RoboDK station: Maoyi_GlueDispensing_PM3.rdk

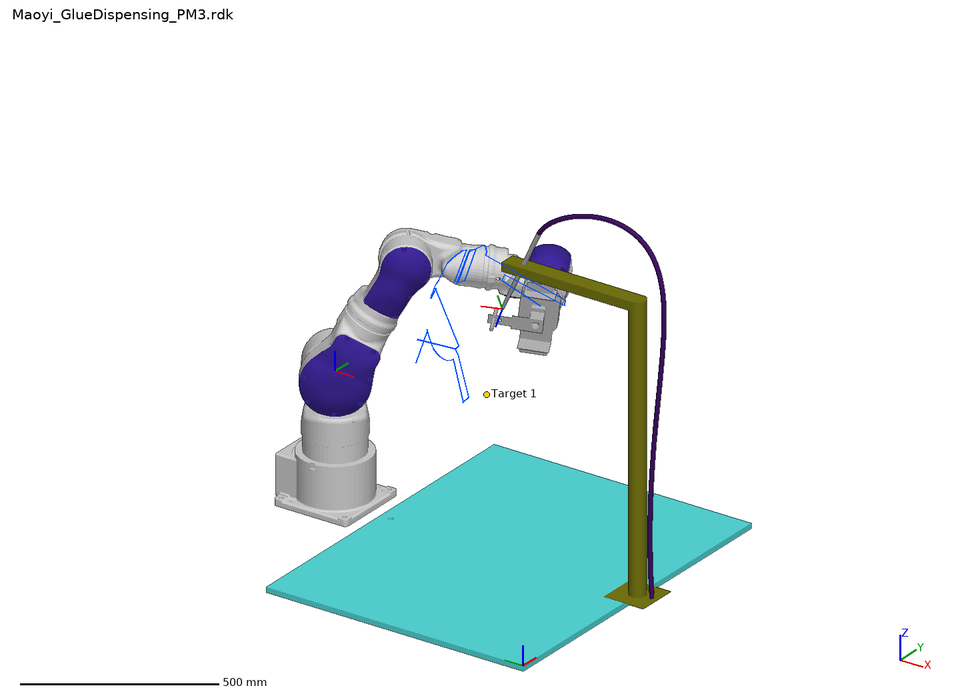
[picture v0: the station drawn from its stored meshes, robots at their saved joint values, targets as dots, program paths as lines]
Station Maoyi_GlueDispensing_PM3 (saved by RoboDK 5.2.1). Poses are relative to the parent item; angles as X-Y-Z fixed-axis rotations.
Station parameters (name, value as stored): IO_5, 1, IO_1, 0, IO_2, 0, IO_3, 1, CollisionFreePlanner, Motoman SIA10D, CollisionFreePlanner-Rob Motoman SIA10D
  - frame Motoman SIA10D Base at (0, 0, 360) mm
    - robot Motoman SIA10D: 7 axes, payload 10 kg, reach 720 mm, repeatability 0.1 mm, weight 60 kg
        modified DH rows (alpha deg, a mm, theta deg, d mm): 0, 0, 0, 360; -90, 0, 0, 0; 90, 0, 0, 360; -90, 0, 0, 0; 90, 0, 0, 360; -90, 0, 0, 0; 90, 0, 180, 155
        base shift (0, 0, -360) mm
        joint limits [-180, -110, -170, -135, -180, -110, -180] to [180, 110, 170, 135, 180, 110, 180]; home [0, 0, 0, 90, 0, 0, 0]; saved at [35.072, 29.67, 0, 66.212, -82.383, 96.989, -179.696]
      - tool Suction_cup, TCP at (106, 0, 141) mm, size 171 x 210 x 141 mm, geometry from Suction_cup.step
      - tool Path 1, TCP at (0, 0, 0) mm
    - frame Working plan at (927.5, -500, -365) mm, rotated rx 0 ry 0 rz 90 deg
      - object robot_platform1 at (0, 0, 0) mm, size 1000 x 790 x 15 mm, geometry from robot_platform1.step
      - object Dispensing Tool at (0, 0, 0) mm, rotated rx 90 ry 0 rz 180 deg, size 120 x 1028.7 x 505.5 mm, geometry from Dispensing Tool.step
      - target Target 1 (Cartesian target) at (500, 461.5, 429) mm, rotated rx -180 ry 0 rz -90 deg; joints [0, 0, 0, 90, 0, 90, 0] of Motoman SIA10D
  - frame Glue at (512.5, 0, 678) mm, rotated rx 169 ry -15 rz -130 deg
  - machining project Path 1 Settings: rotZ(0) | rotX(0)*rotY(0) | rotz(0) | onStart | onPathStart | onApproach | onPoint | onRetract | onFinish | SetRPM(%1) | SetTool(%1) | Extruder(%1) | default | default | OutOnMov(%1) | OutOffMov(%1) | onPathFinish | M_RunCode(%1) | WAN Miniport (IPv6)-QoS 
  - program Path (93 instructions, listed below)
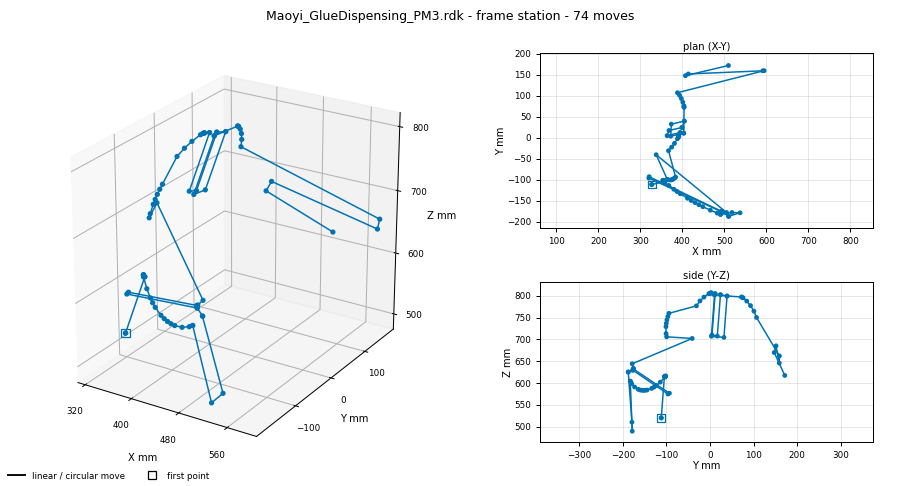
[picture p0: tool path of Maoyi_GlueDispensing_PM3.rdk in frame station, 74 of 74 moves have a stored position in this frame; points joined in program order, loops and branches not executed]

--- program Path (robot Motoman SIA10D) ---
  Smooth(1)
  Set speed (1000.0 mm/s)
  Set Ref.: Glue
  Set Tool: Path 1
  Show Path 1
  MoveJ 1 to (157.11, 29.72, 215.15) mm, rotated rx 0 ry 88 rz 170 deg; joints [-43.735, 4.404, 0, 111.833, 70.327, 95.789, -105.561]
  MoveL 2 to (157.11, 29.72, 215.15) mm, rotated rx 0 ry 88 rz 170 deg; joints [-43.735, 4.404, 0, 111.833, 70.327, 95.789, -105.561]
  MoveL 3 to (157.11, 29.72, 115.15) mm, rotated rx 0 ry 88 rz 170 deg; joints [-39.6, 2.361, 0, 98.055, 73.469, 96.968, -89.206]
  MoveL 4 to (157.11, 29.72, 115.15) mm, rotated rx 0 ry 88 rz 170 deg; joints [-39.6, 2.361, 0, 98.055, 73.469, 96.968, -89.206]
  Set speed (50.0 mm/s)
  MoveL 5 to (157.93, 34.33, 115.15) mm, rotated rx 0 ry 88 rz 170 deg; joints [-39.683, 1.614, 0, 98.657, 73.469, 97.088, -89.089]
  MoveL 6 to (157.93, 34.32, 115.15) mm, rotated rx 0 ry 88 rz 170 deg; joints [-39.683, 1.616, 0, 98.655, 73.469, 97.09, -89.09]
  MoveL 7 to (158.06, 34.91, 115.26) mm, rotated rx -2.73 ry 88 rz 167.24 deg; joints [-39.701, 1.529, 0, 98.739, 73.466, 97.13, -89.188]
  MoveL 8 to (158.06, 34.43, 115.85) mm, rotated rx -18.04 ry 87.9 rz 151.87 deg; joints [-39.727, 1.632, 0, 98.745, 73.448, 97.185, -89.858]
  MoveL 9 to (157.82, 32.09, 117.26) mm, rotated rx -45.21 ry 87.16 rz 124.55 deg; joints [-39.76, 2.054, 0, 98.615, 73.405, 97.245, -91.521]
  MoveL 10 to (154.79, 14.07, 124.94) mm, rotated rx -79.41 ry 79.05 rz 90.27 deg; joints [-39.761, 4.944, 0, 97.388, 73.212, 96.698, -101.87]
  MoveL 11 to (152.01, -2.22, 129.27) mm, rotated rx -83.67 ry 71.55 rz 85.94 deg; joints [-39.66, 7.569, 0, 95.743, 73.132, 96.266, -110.361]
  MoveL 12 to (150.39, -11.66, 130.72) mm, rotated rx -84.8 ry 67.34 rz 84.72 deg; joints [-39.564, 9.1, 0, 94.562, 73.121, 96.077, -114.908]
  MoveL 13 to (148.65, -21.63, 131.47) mm, rotated rx -85.59 ry 63.01 rz 83.78 deg; joints [-39.434, 10.743, 0, 93.127, 73.132, 95.975, -119.417]
  MoveL 14 to (145.06, -41.61, 130.64) mm, rotated rx -86.59 ry 54.07 rz 82.68 deg; joints [-39.109, 13.918, 0, 89.873, 73.23, 95.62, -128.205]
  MoveL 15 to (143.2, -51.74, 128.99) mm, rotated rx -86.92 ry 49.53 rz 82.27 deg; joints [-38.91, 15.538, 0, 87.958, 73.31, 95.519, -132.41]
  MoveL 16 to (141.35, -61.66, 126.55) mm, rotated rx -87.17 ry 45.01 rz 81.92 deg; joints [-38.694, 17.127, 0, 85.908, 73.408, 95.449, -136.437]
  MoveL 17 to (139.52, -71.34, 123.32) mm, rotated rx -87.37 ry 40.49 rz 81.63 deg; joints [-38.462, 18.685, 0, 83.728, 73.521, 95.41, -140.298]
  MoveL 18 to (137.59, -80.96, 119.31) mm, rotated rx -87.53 ry 35.95 rz 81.29 deg; joints [-38.204, 20.28, 0, 81.348, 73.653, 95.468, -144.012]
  MoveL 19 to (134.09, -98.51, 109.2) mm, rotated rx -87.76 ry 26.98 rz 80.87 deg; joints [-37.688, 23.195, 0, 76.452, 73.945, 95.527, -150.939]
  MoveL 20 to (131.11, -113.4, 97.08) mm, rotated rx -87.89 ry 18.43 rz 80.59 deg; joints [-37.184, 25.777, 0, 71.498, 74.251, 95.627, -157.067]
  MoveL 21 to (129.91, -120.19, 89.79) mm, rotated rx -87.94 ry 13.91 rz 80.57 deg; joints [-36.937, 26.977, 0, 68.888, 74.405, 95.615, -160.156]
  Set speed (1000.0 mm/s)
  MoveL 22 to (129.91, -120.19, 89.79) mm, rotated rx -87.94 ry 13.91 rz 80.57 deg; joints [-36.937, 26.977, 0, 68.888, 74.405, 95.615, -160.156]
  MoveL 23 to (79.99, -157.87, 189.79) mm, rotated rx -87.94 ry 13.91 rz 60.22 deg; joints [-33.756, 43.629, 0, 63.422, 72.969, 109.883, -171.1]
  Set speed (1000.0 mm/s)
  MoveL 24 to (73.82, -168.5, 164.19) mm, rotated rx -88 ry 0 rz 60.21 deg; joints [-32.838, 45.387, 0, 56.918, 74.962, 109.853, -179.878]
  MoveL 25 to (127, -133.09, 64.19) mm, rotated rx -88 ry 0 rz 80.21 deg; joints [-36.118, 29.852, 0, 61.258, 74.923, 95.954, -169.241]
  MoveL 26 to (126.52, -133.55, 64.19) mm, rotated rx -88 ry 0 rz 80 deg; joints [-36.071, 30.04, 0, 61.029, 74.968, 96.124, -169.193]
  Set speed (50.0 mm/s)
  MoveL 27 to (129.86, -114.6, 64.19) mm, rotated rx -88 ry 0 rz 80 deg; joints [-36.182, 26.681, 0, 65.29, 74.87, 95.997, -170.098]
  Set speed (1000.0 mm/s)
  MoveL 28 to (129.86, -114.6, 64.19) mm, rotated rx -88 ry 0 rz 80 deg; joints [-36.182, 26.681, 0, 65.29, 74.87, 95.997, -170.098]
  MoveL 29 to (164.2, 55.09, 164.19) mm, rotated rx -88 ry 0 rz 139.98 deg; joints [-27.408, -26.255, 0, 125.061, 62.627, 26.628, -163.821]
  Set speed (1000.0 mm/s)
  MoveL 30 to (161.83, 57.08, 162.05) mm, rotated rx -88 ry -1.39 rz 139.98 deg; joints [-26.439, -26.479, 0, 124.899, 61.136, 25.919, -163.397]
  MoveL 31 to (130.35, -111.61, 62.05) mm, rotated rx -88 ry -1.39 rz 79.98 deg; joints [-36.14, 26.217, 0, 65.529, 74.89, 95.991, -171.263]
  MoveL 32 to (130.13, -111.86, 62.05) mm, rotated rx -88 ry -1.39 rz 79.87 deg; joints [-36.119, 26.314, 0, 65.416, 74.913, 96.083, -171.244]
  Set speed (50.0 mm/s)
  MoveL 33 to (129.74, -112.87, 60.31) mm, rotated rx -88 ry -2.52 rz 79.73 deg; joints [-36.042, 26.592, 0, 64.804, 74.967, 96.19, -172.029]
  MoveL 34 to (128.05, -120.15, 47.08) mm, rotated rx -87.96 ry -10.74 rz 79.49 deg; joints [-35.616, 28.352, 0, 60.515, 75.241, 96.377, -177.685]
  MoveL 35 to (145.22, 103.16, 33.99) mm, rotated rx -87.89 ry -18.35 rz 159.26 deg; joints [4.953, -25.059, 0, 105.149, -46, 38.82, -71.346]
  MoveL 36 to (173.24, 45.66, 26.51) mm, rotated rx -87.83 ry -22.55 rz 139.09 deg; joints [-23.233, -19.082, 0, 99.7, 35.021, 35.81, -154.435]
  MoveL 37 to (174.4, 44.13, 18.62) mm, rotated rx -87.76 ry -26.89 rz 138.83 deg; joints [-23.305, -18.367, 0, 98.004, 34.452, 36.71, -158.019]
  MoveL 38 to (175.18, 42.9, 2.05) mm, rotated rx -87.53 ry -35.86 rz 138.47 deg; joints [-22.792, -17.072, 0, 94.566, 32.168, 38.176, -164.291]
  MoveL 39 to (174.85, 42.8, -6.35) mm, rotated rx -87.37 ry -40.39 rz 138.22 deg; joints [-22.369, -16.422, 0, 92.824, 30.913, 38.891, -167.337]
  MoveL 40 to (174.01, 43.13, -14.72) mm, rotated rx -87.18 ry -44.91 rz 137.93 deg; joints [-21.813, -15.791, 0, 91.098, 29.531, 39.567, -170.259]
  MoveL 41 to (172.66, 43.88, -23) mm, rotated rx -86.92 ry -49.44 rz 137.58 deg; joints [-21.129, -15.181, 0, 89.395, 28.03, 40.207, -173.075]
  MoveL 42 to (170.88, 44.82, -31.14) mm, rotated rx -86.6 ry -53.97 rz 137.09 deg; joints [-20.401, -14.554, 0, 87.701, 26.629, 40.876, -175.981]
  MoveL 43 to (139.27, 102.19, -46.62) mm, rotated rx -85.6 ry -62.93 rz 155.93 deg; joints [6.632, -17.369, 0, 88.025, -40.603, 46.772, -123.836]
  MoveL 44 to (131.48, 104.56, -60.31) mm, rotated rx -83.7 ry -71.46 rz 153.89 deg; joints [8.407, -15.487, 0, 84.78, -41.554, 48.903, -131.896]
  MoveL 45 to (122.84, 107.36, -71.41) mm, rotated rx -79.42 ry -79.04 rz 149.5 deg; joints [10.261, -13.751, 0, 82.013, -42.758, 50.843, -138.763]
  MoveL 46 to (111.97, 111.11, -81.89) mm, rotated rx -51.66 ry -86.77 rz 121.72 deg; joints [12.505, -11.85, 0, 79.233, -44.447, 52.98, -145.776]
  MoveL 47 to (108.77, 112.18, -84.01) mm, rotated rx -18.09 ry -87.9 rz 88.11 deg; joints [13.101, -11.387, 0, 78.632, -44.881, 53.454, -147.298]
  MoveL 48 to (107.24, 112.71, -84.62) mm, rotated rx -2.74 ry -88 rz 72.74 deg; joints [13.386, -11.208, 0, 78.443, -45.117, 53.644, -147.638]
  MoveL 49 to (106.3, 113.05, -84.72) mm, rotated rx 0 ry -88 rz 70 deg; joints [13.568, -11.125, 0, 78.393, -45.294, 53.742, -147.557]
  MoveL 50 to (106.3, 113.04, -84.72) mm, rotated rx 0 ry -88 rz 70 deg; joints [13.565, -11.126, 0, 78.393, -45.289, 53.739, -147.561]
  MoveL 51 to (97.54, 116.23, -84.72) mm, rotated rx 0 ry -88 rz 70 deg; joints [15.2, -10.452, 0, 78.145, -46.895, 54.532, -145.889]
  Set speed (1000.0 mm/s)
  MoveL 52 to (97.54, 116.23, -84.72) mm, rotated rx 0 ry -88 rz 70 deg; joints [15.2, -10.452, 0, 78.145, -46.895, 54.532, -145.889]
  MoveL 53 to (97.54, 116.23, 15.28) mm, rotated rx 0 ry -88 rz 70 deg; joints [15.484, -19.399, 0, 100.403, -55.741, 46.38, -132.19]
  Set speed (1000.0 mm/s)
  MoveL 54 to (85.1, 120.76, 15.28) mm, rotated rx 0 ry -88 rz 70 deg; joints [17.975, -18.21, 0, 99.985, -57.959, 48.02, -129.475]
  MoveL 55 to (85.1, 120.76, -84.72) mm, rotated rx 0 ry -88 rz 70 deg; joints [17.413, -9.433, 0, 77.725, -48.993, 55.654, -143.671]
  MoveL 56 to (85.1, 120.76, -84.72) mm, rotated rx 0 ry -88 rz 70 deg; joints [17.413, -9.433, 0, 77.725, -48.993, 55.654, -143.671]
  Set speed (50.0 mm/s)
  MoveL 57 to (69.68, 126.37, -84.72) mm, rotated rx 0 ry -88 rz 70 deg; joints [19.984, -8.074, 0, 77.093, -51.323, 57.027, -141.157]
  Set speed (1000.0 mm/s)
  MoveL 58 to (69.68, 126.37, -84.72) mm, rotated rx 0 ry -88 rz 70 deg; joints [19.984, -8.074, 0, 77.093, -51.323, 57.027, -141.157]
  MoveL 59 to (69.68, 126.37, 15.28) mm, rotated rx 0 ry -88 rz 70 deg; joints [20.844, -16.633, 0, 99.36, -60.324, 49.973, -126.461]
  Set speed (1000.0 mm/s)
  MoveL 60 to (92.36, 108.64, 15.28) mm, rotated rx 0 ry -88 rz 50 deg; joints [2.349, -20.756, 0, 100.584, -8.82, 30.436, -175.631]
  MoveL 61 to (92.36, 108.64, -84.72) mm, rotated rx 0 ry -88 rz 50 deg; joints [3.664, -11.631, 0, 78.327, -8.266, 43.611, -176.796]
  MoveL 62 to (92.36, 108.64, -84.72) mm, rotated rx 0 ry -88 rz 50 deg; joints [3.664, -11.631, 0, 78.327, -8.266, 43.611, -176.796]
  Set speed (50.0 mm/s)
  MoveL 63 to (44.75, 148.58, -84.72) mm, rotated rx 0 ry -88 rz 50 deg; joints [16.892, -10.157, 0, 78.01, -25.535, 46.077, -159.742]
  MoveL 64 to (44.81, 148.57, -84.72) mm, rotated rx 0 ry -88 rz 49.98 deg; joints [16.868, -10.165, 0, 78.014, -25.474, 46.063, -159.794]
  MoveL 65 to (42.16, 151, -83.29) mm, rotated rx 33.09 ry -87.61 rz 16.77 deg; joints [17.555, -10.197, 0, 78.31, -26.267, 46.069, -160.234]
  MoveL 66 to (35.52, 156.94, -75.87) mm, rotated rx 74.88 ry -82.31 rz -25.13 deg; joints [19.397, -10.599, 0, 79.943, -28.959, 45.773, -163.445]
  MoveL 67 to (28.54, 163.33, -65.6) mm, rotated rx 82.26 ry -74.98 rz -32.67 deg; joints [21.369, -11.199, 0, 82.176, -31.987, 45.298, -167.527]
  MoveL 68 to (22.18, 169.3, -52.82) mm, rotated rx 84.94 ry -66.7 rz -35.5 deg; joints [23.237, -11.987, 0, 84.916, -35.114, 44.646, -172.24]
  MoveL 69 to (17.09, 174.28, -37.95) mm, rotated rx 86.24 ry -57.85 rz -36.97 deg; joints [24.85, -12.95, 0, 88.063, -38.171, 43.818, -177.473]
  MoveL 70 to (-172.68, 44.47, -21.93) mm, rotated rx 86.96 ry -48.86 rz 42.13 deg; joints [28.642, 62.203, 0, 5.637, -97.473, 108.983, -172.895]
  MoveL 71 to (-174.72, 43.55, -5.38) mm, rotated rx 87.39 ry -39.86 rz 41.5 deg; joints [28.755, 56.395, 0, 19.451, -94.687, 109.93, -173.467]
  MoveL 72 to (-48.92, 173.48, 12.49) mm, rotated rx 87.69 ry -30.23 rz -19 deg; joints [37.01, -1.889, 0, 90.072, -69.478, 62.199, -172.135]
  MoveL 73 to (-45.54, 172.88, 29.51) mm, rotated rx 87.86 ry -20.88 rz -19.41 deg; joints [37.157, -3.194, 0, 93.766, -70.706, 61.52, -178.892]
  MoveL 74 to (-140.59, 105.65, 45.91) mm, rotated rx 87.96 ry -11.44 rz 20.28 deg; joints [35.072, 29.67, 0, 66.212, -82.383, 96.989, -179.696]
  Set speed (1000.0 mm/s)
